INTERFACE I_UDINT EXTENDS I_Datatype

PROPERTY PUBLIC Value : REFERENCE TO UDINT
GET
END_GET
END_PROPERTY

END_INTERFACE

(* stored: Version 1.1.0.1, ProductVersion 3.1.4024.15
   Itf I_UDINT: Id {478de083-5c4f-080c-34de-b24804f021cb}
   Property Value: Id {1c6665d8-c1f7-01fe-23df-696d80f8fe7e}
   Get Get: Id {21a02be0-3565-0e25-2109-223ae50c011c} *)
